PROGRAM MAIN_Fast
VAR_INPUT
END_VAR
VAR
END_VAR
VAR_OUTPUT	
END_VAR

// fast stuff here..

fbModul001.M_Fast();

END_PROGRAM

(* stored: Version 1.1.0.1
   POU MAIN_Fast: Id {59b841e9-8296-4be5-ae67-17d2cafdeea1}, SpecialFunc None *)
